// TIA Portal V20 export
TYPE "LER_typeGearInInterface"
// stored: Access Published
   STRUCT
      gearInOn : Bool;
      gearInOff : Bool;
      monitoring : "LER_typeGearInMonitoring";
   END_STRUCT;
END_TYPE
